// TIA Portal V17 export
// export: Created 2024-10-17T14:16:20.2364585Z, ExportSetting WithDefaults, DisplayName Totally Integrated Automation Portal, DisplayVersion V17 Update 4, DisplayName TIA Portal Openness, DisplayVersion V17 Update 4, DisplayName TIA Portal Version Control Interface, DisplayVersion V17, DisplayName SINAMICS Startdrive Advanced, DisplayVersion V17 Update2, DisplayName SINAMICS Startdrive G130, G150, S120, S150, SINAMICS MV, S210, DisplayVersion V17 Update2, DisplayName SINAMICS Startdrive G110M, G120, G120C, G120D, G120P, G115D, DisplayVersion V17 Update2, DisplayName STEP 7 Professional, DisplayVersion V17 Update 4, DisplayName STEP 7 Safety, DisplayVersion V17, DisplayName WinCC Advanced / Unified PC, DisplayVersion V17 Update 4
TYPE "LPMLV2022_typeConfiguration"
TITLE = LPMLV2022_typeConfiguration
// Support: tech.team.motioncontrol@siemens.com
// stored: IsFailsafeCompliant false
   STRUCT
      EnabledModesCfg : DWord := 16#0000_01FE;   // Bit locations within the DWORD represent Mode numbers. A value of 1 in a bit location [0-31] indicates that the corresponding Mode number is enabled. Mode 0 is an Invalid Mode, therefore bit 0 is unused
      DisabledStatesCfg : Array[0.."LPMLV2022_MAX_MODES_UPPER_LIM"] of DWord;   // The array index represents the Mode number. Bit locations within the DWORD value represent State numbers. A value of 1 in a bit location indicates that the corresponding state number is disabled. State 0 is an Undefined State, therefore bit 0 is unused
      ModeTransitionCfg : Array[0.."LPMLV2022_MAX_MODES_UPPER_LIM"] of DWord;   // The array index represents the Mode number. Bit locations within the DWORD value represent State numbers. A value of 1 in a bit location indicates that a mode transition from the corresponding state number is allowed
      holdCmdCfg : DWord := 16#0000_0060;   // Bit locations within the DWORD value represent State numbers. A value of 1 in a bit location indicates that the Hold control command is taken into account in the corresponding state. Note: a state change is only performed if the Holding/Held states are not disabled. The 'holdCmdCfg' can only be activated for the following states: Idle, Starting, Execute, Completing, Completed, Suspending, Suspended, Unsuspending, Unholding
      completeCmdCfg : DWord := 16#0000_0860;   // Bit locations within the DWORD value represent State numbers. A value of 1 in a bit location indicates that the Complete control command is taken into account in the corresponding state. Note: a state change is only performed if the Completing/Completed states are not disabled. The 'completeCmdCfg' can only be activated for the following states: Execute, Suspended, Held
   END_STRUCT;
   // ModeTransitionCfg[1..31] := 16#0000_0214;
END_TYPE
